(* CoDeSys 2.3.9.35 project: easynet_XV200Masteraus EC4P.pro *)
(* Libraries: SysLibRtc.lib*29.9.06 14:48:48, SysLibEasyNet.lib*30.6.08 13:43:32, easyNet.lib*8.2.21 14:46:37, Util.lib 3.7.08 07:33:54, SysLibSockets.lib 3.7.08 07:33:54, SysLibTasks.lib 3.7.08 07:33:54, SysLibFile.lib 29.9.06 14:48:48, SysLibPlcCtrl.lib 29.9.06 14:48:48, Standard.lib 5.4.06 14:34:00, SYSLIBCALLBACK.LIB 27.8.10 15:11:00 *)

(* PLC configuration (modules and I/O channels)
Configuration XC-CPU201-EC512K-8DI-6DO-XV [Root] node -1, in %IB0 out %QB0 {PXC101_1 = WARMSTART; PXC101INT = 0; PXC101INT = 0; PXC101INT = 0; PXC101INT = 0; PX101PARWORD = 0; PX101PARWORD = 0; PX101PARWORD = 0; PXC101ROUTING1 = 125KBaud; PXC101ROUTING2 = 127; PXC101INT = 0; PXC101INT = 0; PXC101ROUTING3 = 1; PXC101ROUTING4 = 0; PXC101_4 = Default; PXC101_5 = Default; PXC101_6 = Default; PXC101_7 = Default; PXC101_8 = None}
  AT %IB0 [LocalInput] Local Inputs/Counter
  AT %IX1.0 [LokalBitin201] State
  AT %IX1.1 [LokalBitin201] N0
  AT %IX1.2 [LokalBitin201] N1
  AT %IX1.3 [LokalBitin201] Error
  AT %IX1.4 [LokalBitin201] Referencing activated
  AT %IW2 [WordInput] Counter-Value Low-Word
  AT %IW4 [WordInput] Counter-Value High-Word
  AT %QB0 [LocalOutput] Local Outputs
  AT %QX1.0 [LokalBitout201] Reference Window
  AT %QX1.1 [LokalBitout201] Reset Counter0
  AT %QX1.2 [LokalBitout201] Reset Counter1
  AT %QX1.3 [LokalBitout201] N0 Quit
  AT %QX1.4 [LokalBitout201] N1 Quit
  AT %QX1.5 [LokalBitout201] Error Quit
  AT %QX1.6 [LokalBitout201] 32BitCounter/Counter0 Enable
  AT %QX1.7 [LokalBitout201] Counter1 Enable
  Non Display [NoDisp] node 0, in %IB6 out %QB2
    EMPTY-SLOT [XIOC_EMPTY] node 0, in %IB6 out %QB2
    EMPTY-SLOT [XIOC_EMPTY] node 1, in %IB6 out %QB2
    EMPTY-SLOT [XIOC_EMPTY] node 2, in %IB6 out %QB2
    EMPTY-SLOT [XIOC_EMPTY] node 3, in %IB6 out %QB2
    EMPTY-SLOT [XIOC_EMPTY] node 4, in %IB6 out %QB2
    EMPTY-SLOT [XIOC_EMPTY] node 5, in %IB6 out %QB2
    EMPTY-SLOT [XIOC_EMPTY] node 6, in %IB6 out %QB2
    EMPTY-SLOT [XIOC_EMPTY] node 7, in %IB6 out %QB2
    EMPTY-SLOT [XIOC_EMPTY] node 8, in %IB6 out %QB2
    EMPTY-SLOT [XIOC_EMPTY] node 9, in %IB6 out %QB2
    EMPTY-SLOT [XIOC_EMPTY] node 10, in %IB6 out %QB2
    EMPTY-SLOT [XIOC_EMPTY] node 11, in %IB6 out %QB2
    EMPTY-SLOT [XIOC_EMPTY] node 12, in %IB6 out %QB2
    EMPTY-SLOT [XIOC_EMPTY] node 13, in %IB6 out %QB2
    EMPTY-SLOT [XIOC_EMPTY] node 14, in %IB6 out %QB2
*)

(* Global variable list: Simulation_IO *)
VAR_GLOBAL
	I1:BOOL;
	I2:BOOL;
	I3:BOOL;
	I4:BOOL;
	I5:BOOL;
	I6:BOOL;
	I7:BOOL;
	I8:BOOL;
	I9:BOOL;
	I10:BOOL;
	I11:BOOL;
	I12:BOOL;
	I13:BOOL;
	I14:BOOL;
	I15:BOOL;
	I16:BOOL;

	Q1:BOOL;
	Q2:BOOL;
	Q3:BOOL;
	Q4:BOOL;
	Q5:BOOL;
	Q6:BOOL;
	Q7:BOOL;
	Q8:BOOL;

END_VAR

(* POU PLC_PRG, IL *)
PROGRAM PLC_PRG
VAR
	(********************************************************************************************************)
	(* easy_net_Sychronisation der Geräteuhr															*)
	(********************************************************************************************************)
	dtRtcClock					: DT;
	SysUhr					: BOOL;
	udiSecondsSince1970	: UDINT;
	udiSecondsOfWeek		: UDINT;
	xNotFirstCycle				: BOOL;
	TON1						: TON;

	(********************************************************************************************************)
	(* Put und Get *)
	(********************************************************************************************************)
	Put_1						: Put;
	Put_4						: Put;
	Get_1 						: Get;
	Get_2 						: Get;

	(********************************************************************************************************)
	(* Für Visualisierung																					*)
	(********************************************************************************************************)
	I1_Visu					: BOOL;
	I2_Visu					: BOOL;

	PT_Nr_Put1				: BYTE:=1;
	I1_1						: DINT:=10000;
	T_1						: BOOL:=TRUE;

	PT_Nr_Put4				: BYTE:=4;
	I1_4						: DINT:=40000;
	T_4						: BOOL:=TRUE;

	GT_Nr_1					: BYTE:=1;
	NET_ID_1					: BYTE:=1;
	PT_Nr_Get1				: BYTE:=1;

	GT_Nr_2					: BYTE:=2;
	NET_ID_2					: BYTE:=1;
	PT_Nr_Get2				: BYTE:=4;
END_VAR
	(**********************************************************************************************************************************************)
	(* Der Aufruf der easy_net_manage Programm																							   *)
	(**********************************************************************************************************************************************)
	CAL		easy_net_manage()

	(**********************************************************************************************************************************************)
	(* Der Aufruf der easy_net_Sychronisation der Geräteuhr																				   *)
	(**********************************************************************************************************************************************)
	LD		TRUE
	SysRtcGetTime
	ST		dtRtcClock
	DT_TO_UDINT
	ST		udiSecondsSince1970
	MOD		86400
	ST		udiSecondsOfWeek
	EQ		43200
	ST		myEASY_NET_MAIN.SND.xStartClockSynchronisation

	(**********************************************************************************************************************************************)
	(* an NET-ID2 zustand Bits 1und 2 senden																								   *)
	(**********************************************************************************************************************************************)
	LD		I1_Visu
	OR		I1
	ST		NET_2SN[1]

	LD		I2_Visu
	OR		I2
	ST		NET_2SN[2]

	(**********************************************************************************************************************************************)
	(* von NET-ID2 zustand Bits 1und 2 empfangen																							   *)
	(**********************************************************************************************************************************************)
	LD		NET_2RN[1]
	ST		Q1
	LD		NET_2RN[2]
	ST		Q2

	(**********************************************************************************************************************************************)
	(* Daten versenden an NET-ID1 mit Put1und Put4																						   *)
	(*Die Übertragung wird einmalig durch eine positive Flanke am Baustein-Eingang T_ gestartet. 									   *)
	(**********************************************************************************************************************************************)
	CAL		Put_1(
	PT_Nr:=PT_Nr_Put1,		(* Modulnummer eingabe der zu sendenden Daten PUT *)
	I1:=I1_1,					(* Nutzdaten (4Byte) *)
	T_:=,						(* Ein Wechsel von FALSE auf TRUE startet das Versenden von eingetragenen Daten.*)
	Q1=> ,						(* Ein Wechsel von FALSE auf TRUE startet das Versenden von eingetragenen Daten.*)
	AC=> ,						(* FALSE =	Das Versenden der Daten wurde erfolgreich abgeschlossen.*)
	E1=> )						(* FALSE =	Der Sendebaustein ist frei. Ein neuer Sendeauftrag kann durch setzten von T_ abgesetzt werden.*)

	CAL		Put_4(
	PT_Nr:=PT_Nr_Put4,		(* Modulnummer eingabe der zu sendenden Daten PUT *)
	I1:=I1_4,					(* Nutzdaten (4Byte) *)
	T_:=,						(* Ein Wechsel von FALSE auf TRUE startet das Versenden von eingetragenen Daten.*)
	Q1=> ,						(* Ein Wechsel von FALSE auf TRUE startet das Versenden von eingetragenen Daten.*)
	AC=> ,						(* FALSE =	Das Versenden der Daten wurde erfolgreich abgeschlossen.*)
	E1=> )						(* FALSE =	Der Sendebaustein ist frei. Ein neuer Sendeauftrag kann durch setzten von T_ abgesetzt werden.*)

	(**********************************************************************************************************************************************)
	(* Daten auslesen von NET-ID1 mit Get1 und Get4																						   *)
	(**********************************************************************************************************************************************)
	CAL		Get_1(
	GT_Nr:=GT_Nr_1,			(* Get Bausteinnummert *)
	NET_ID:=NET_ID_1,		(* Net-ID des Teilnehmers eingetragen, der das zu empfangende GET - Telegramm aussendet.*)
	PT_Nr:=PT_Nr_Get1,		(* Modulnummer eingabe der zu empfangenden Daten GET *)
	QV=> ,						(* Der zuletzt empfangene Stand der Nutzdaten *)
	Q1=> )						(* TRUE:Erster Lesezugriff auf neu eingetroffene Daten.*)

	CAL		Get_2(
	GT_Nr:=GT_Nr_2,			(* Get Bausteinnummert *)
	NET_ID:=NET_ID_2,		(* Net-ID des Teilnehmers eingetragen, der das zu empfangende GET - Telegramm aussendet.*)
	PT_Nr:=PT_Nr_Get2,		(* Modulnummer eingabe der zu empfangenden Daten GET *)
	QV=> ,						(* Der zuletzt empfangene Stand der Nutzdaten *)
	Q1=> )						(* TRUE:Erster Lesezugriff auf neu eingetroffene Daten.*)

	(**********************************************************************************************************************************************)
	(*Programm Ende																														   *)
	(**********************************************************************************************************************************************)
END_PROGRAM

(* Visualisation Beispiel_Netvisu
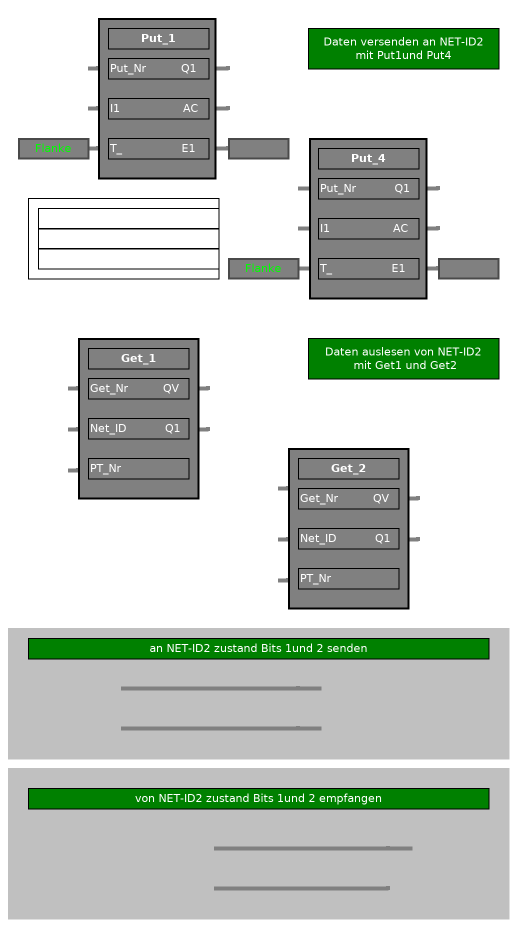
group at (20,10)-(521,921)
  rectangle at (220,130)-(281,151): text "aktiv"; invisible if PLC_PRG.Put_1.E1; alarm colour if NOT(PLC_PRG.Put_1.E1)
  rectangle at (300,20)-(491,61): text "Daten versenden an NET-ID2 / mit Put1und Put4"
  rounded rectangle at (100,50)-(201,71): text "Put_Nr          Q1"
  rounded rectangle at (100,90)-(201,111): text "I1                  AC"
  rounded rectangle at (100,130)-(201,151): text "T_                 E1"
  rectangle at (220,130)-(281,151): invisible if PLC_PRG.Put_1.T_
  rectangle at (10,130)-(81,151): text "Flanke"; alarm colour if PLC_PRG.Put_1.T_; taps PLC_PRG.Put_1.T_
  rectangle at (100,20)-(201,41): text "Put_1"
  rounded rectangle at (310,140)-(411,161): text "Put_4"
  rounded rectangle at (310,170)-(411,191): text "Put_Nr           Q1"
  rounded rectangle at (310,210)-(411,231): text "I1                  AC"
  rounded rectangle at (310,250)-(411,271): text "T_                 E1"
  rectangle at (220,250)-(291,271): text "Flanke"; alarm colour if PLC_PRG.Put_4.T_; taps PLC_PRG.Put_4.T_
  rectangle at (430,250)-(491,271): text "aktiv"; invisible if PLC_PRG.Put_4.E1; alarm colour if NOT(PLC_PRG.Put_4.E1)
  rectangle at (430,250)-(491,271): invisible if PLC_PRG.Put_4.T_
  group at (20,190)-(211,271)
    rectangle at (10,10)-(191,31): text "Die Übertragung wird einmalig"
    rectangle at (10,30)-(191,51): text "durch eine positive Flanke am"
    rectangle at (10,50)-(191,71): text "Baustein-Eingang T_ gestartet."
  rectangle at (300,330)-(491,371): text "Daten auslesen von NET-ID2 / mit Get1 und Get2"
  rounded rectangle at (290,450)-(391,471): text "Get_2"
  rounded rectangle at (290,480)-(391,501): text "Get_Nr          QV"
  rounded rectangle at (290,520)-(391,541): text "Net_ID           Q1"
  rounded rectangle at (290,560)-(391,581): text "PT_Nr"
  rounded rectangle at (80,340)-(181,361): text "Get_1"
  rounded rectangle at (80,370)-(181,391): text "Get_Nr          QV"
  rounded rectangle at (80,410)-(181,431): text "Net_ID           Q1"
  rounded rectangle at (80,450)-(181,471): text "PT_Nr"
  rectangle at (20,630)-(481,651): text "an NET-ID2 zustand Bits 1und 2 senden"
  rectangle at (20,780)-(481,801): text "von NET-ID2 zustand Bits 1und 2 empfangen"
35 more shapes without text or variables
*)

(* Visualisation net_state_use
embedded screen at (40,30)-(641,321): net_state
*)
